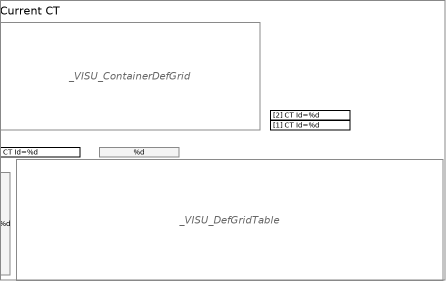
VISUALIZATION _VISU_CT_Details  // 446x281
VAR_IN_OUT
  mInst : FB_WorkerDefGrid;
END_VAR
    Frame (0,22 260x108)
        shows _VISU_ContainerDefGrid(m_Inst := mInst._pAttachedCt^)
    Frame (16,159 427x122)
        shows _VISU_DefGridTable(m_Inst := mInst._pAttachedCt^.fBImageDeformation, m_row_start := mInst.nGridRowStart, m_col_start := mInst.nGridColStart)
    Scrollbar (99,147 80x10), "%d", text variable: mInst.nGridColStart
        p2245068023: mInst._pAttachedCt^.fBImageDeformation.nMAX_ROWS_DEFGRID-2
        p1057716461: mInst.nGridColStart
    Scrollbar (0,172 10x103), "%d", text variable: mInst._pAttachedCt^.sContainer.iId
        p2245068023: mInst._pAttachedCt^.fBImageDeformation.nMAX_ROWS_DEFGRID
        p1057716461: mInst.nGridRowStart
    Label (-3,1 150x20), "Current CT"
    Rectangle (0,147 80x10), "CT Id=%d", text variable: mInst._pAttachedCt^.sContainer.iId
    Rectangle (270,120 80x10), "[1] CT Id=%d", text variable: mInst._pAttachedCTList[1]^.sContainer.iId, input disabled if: mInst._pAttachedCTList[1] = 0
    Rectangle (270,110 80x10), "[2] CT Id=%d", text variable: mInst._pAttachedCTList[1]^.sContainer.iId, invisible if: mInst._pAttachedCTList[2] = 0, input disabled if: mInst._pAttachedCTList[1] = 0
END_VISUALIZATION

(* stored: Version 1.1.0.1, ProductVersion 3.1.4024.11
   Visu _VISU_CT_Details: Id {d9b485fc-6da0-4633-b9c6-9432006ab12a} *)
